// TIA Portal project "conveyor-push-sort" (V19)

(* hardware
DEVICE "S7-1200 station_1"  S7-1200 Station
   slot 0: "Rack_0"  S7-1200 Rack  Rack  V1.0
   slot 1: "PLC_1"  CPU 1214C AC/DC/Rly  6ES7 214-1BG40-0XB0  V4.2
   slot 3: "AQ 1x12BIT_1"  AQ1 signal board  6ES7 232-4HA30-0XB0  V1.0
*)

// ===== PLC "PLC_1"  CPU 1214C AC/DC/Rly =====

VAR_GLOBAL   // PLC tag table "Default tag table"
   "M_Start_LastState_Negative" AT %M11.1 : Bool;
   "M_Running" AT %M11.3 : Bool;
   "M_Push" AT %M11.4 : Bool;
   "M_Start_OneShot_Negative" AT %M11.2 : Bool;
   "M_MetalSensor_LastState_Positive" AT %M11.5 : Bool;
END_VAR

VAR_GLOBAL   // PLC tag table "ConveyorInput"
   "B1_FeederRetracted" AT %I0.2 : Bool;
   "B2_FeederExtended" AT %I0.3 : Bool;
   "B5_ColorSensor_IsWhite" AT %I0.6 : Bool;
   "B6_AtConveyorEnd" AT %I0.7 : Bool;
   "B4_MetalSensor" AT %I0.4 : Bool;
END_VAR

VAR_GLOBAL   // PLC tag table "ConveyorOutput"
   "Y1A_FeederExtend" AT %Q0.3 : Bool;
   "Y1B_FeederRetract" AT %Q0.2 : Bool;
   "B3_PusherRetracted" AT %I0.5 : Bool;
   "M1_ConveyorMove" AT %Q0.4 : Bool;
   "Y2_PusherExtend" AT %Q0.5 : Bool;
END_VAR

VAR_GLOBAL   // PLC tag table "ArmInput"
   "B8_ArmOverTruck" AT %I1.0 : Bool;
   "B7_ArmOverConveyor" AT %I1.1 : Bool;
   "B9_ArmIsDown" AT %I1.2 : Bool;
END_VAR

VAR_GLOBAL   // PLC tag table "OperatorPanel"
   "S1_Start" AT %I0.0 : Bool;   // NO
   "S2_Stop" AT %I0.1 : Bool;   // NO
   "P1_LightGreen" AT %Q0.0 : Bool;
   "P2_LightYellow" AT %Q0.1 : Bool;
END_VAR

VAR_GLOBAL   // PLC tag table "ArmOutput"
   "Y6_ArmFromTruckToConveyor" AT %Q0.6 : Bool;
   "Y4_LowerArm" AT %Q0.7 : Bool;
   "Y5_GripperPressureOn" AT %Q1.0 : Bool;
   "Y3_EnableBlackTruck" AT %Q1.1 : Bool;
   "B10_WhiteTruckActive" AT %I1.3 : Bool;
END_VAR

TYPE "ItemRecord"
   STRUCT
      AccumulatedTime : Time;
      Active : Bool;
   END_STRUCT;
END_TYPE

DATA_BLOCK "DB_Settings"   // DB2
{ S7_Optimized_Access := 'TRUE' }
VERSION : 0.1
   VAR
      FeederDelay : Time := T#100ms;
      ArmPickDelay : Time := T#120ms;
      ArmPlaceDelay : Time := T#200ms;
   END_VAR
BEGIN
END_DATA_BLOCK

DATA_BLOCK "DB_ArmSafeStopSteps"   // DB5
{ S7_Optimized_Access := 'TRUE' }
VERSION : 0.1
   VAR
      MovedOverConveyor : Bool;
      Lowered : Bool;
      Released : Bool;
      Lifted : Bool;
   END_VAR
BEGIN
END_DATA_BLOCK

DATA_BLOCK "DB_ItemTracking"   // DB6
{ S7_Optimized_Access := 'TRUE' }
VERSION : 0.1
   VAR
      ItemList : Array[0..5] of "ItemRecord";
      PrevScanTime : DTL;
      CurrentTime : DTL;
      DeltaTime : Time;
      UntrackedItems : UInt;
      ThresholdTime : Time := T#700ms;
   END_VAR
BEGIN
END_DATA_BLOCK

// folder: System blocks/Program resources

DATA_BLOCK "IEC_Timer_0_DB"   // DB1
{ S7_Optimized_Access := 'TRUE' }
AUTHOR : Simatic
FAMILY : IEC
NAME : IEC_TMR
VERSION : 1.0
// stored: InstanceOfName IEC_TIMER
"IEC_TIMER"
BEGIN
END_DATA_BLOCK

DATA_BLOCK "IEC_Timer_0_DB_1"   // DB3
{ S7_Optimized_Access := 'TRUE' }
AUTHOR : Simatic
FAMILY : IEC
NAME : IEC_TMR
VERSION : 1.0
// stored: InstanceOfName IEC_TIMER
"IEC_TIMER"
BEGIN
END_DATA_BLOCK

DATA_BLOCK "IEC_Timer_0_DB_3"   // DB4
{ S7_Optimized_Access := 'TRUE' }
AUTHOR : Simatic
FAMILY : IEC
NAME : IEC_TMR
VERSION : 1.0
// stored: InstanceOfName IEC_TIMER
"IEC_TIMER"
BEGIN
END_DATA_BLOCK

DATA_BLOCK "IEC_Timer_0_DB_2"   // DB7
{ S7_Optimized_Access := 'TRUE' }
AUTHOR : Simatic
FAMILY : IEC
NAME : IEC_TMR
VERSION : 1.0
// stored: InstanceOfName IEC_TIMER
"IEC_TIMER"
BEGIN
END_DATA_BLOCK

// folder: (top level)

FUNCTION "FC_Conveyor" : Void   // FC1, LAD
{ S7_Optimized_Access := 'TRUE' }
VERSION : 0.1
   VAR_TEMP
      i : Int;
      err : Int;
      CurrentTime : DTL;
   END_VAR
   VAR_TEMP   // added for the SCL form of the ladder/FBD networks
      _w1 : Bool;
   END_VAR
BEGIN

REGION Network 1 (SCL)
   // Track items
   IF "DB_ItemTracking".UntrackedItems > 0 THEN
       FOR #i := 0 TO 5 DO
           IF NOT "DB_ItemTracking".ItemList[#i].Active THEN
               "DB_ItemTracking".ItemList[#i].Active := TRUE;
               "DB_ItemTracking".UntrackedItems := "DB_ItemTracking".UntrackedItems - 1;
           END_IF;

           // If more items remain untracked, continue filling slots
           IF "DB_ItemTracking".UntrackedItems = 0 THEN
               EXIT;
           END_IF;
       END_FOR;
   END_IF;
END_REGION

REGION Network 2 (SCL)
   // Push items that approach pusher based on travel time
   #err := RD_SYS_T("DB_ItemTracking".CurrentTime);

   "DB_ItemTracking".DeltaTime := T_DIFF(IN1:="DB_ItemTracking".CurrentTime,IN2:="DB_ItemTracking".PrevScanTime);
   "DB_ItemTracking".PrevScanTime := "DB_ItemTracking".CurrentTime;

   IF "M1_ConveyorMove" THEN
       FOR #i := 0 TO 5 DO
           IF "DB_ItemTracking".ItemList[#i].Active THEN

               "DB_ItemTracking".ItemList[#i].AccumulatedTime :=
               "DB_ItemTracking".ItemList[#i].AccumulatedTime + "DB_ItemTracking".DeltaTime;

               IF "DB_ItemTracking".ItemList[#i].AccumulatedTime >= "DB_ItemTracking".ThresholdTime THEN
                   "M_Push" := TRUE;
                   "DB_ItemTracking".ItemList[#i].Active := FALSE;
                   "DB_ItemTracking".ItemList[#i].AccumulatedTime := T#0s;
               END_IF;
           END_IF;
       END_FOR;
   END_IF;
END_REGION

REGION Network 3
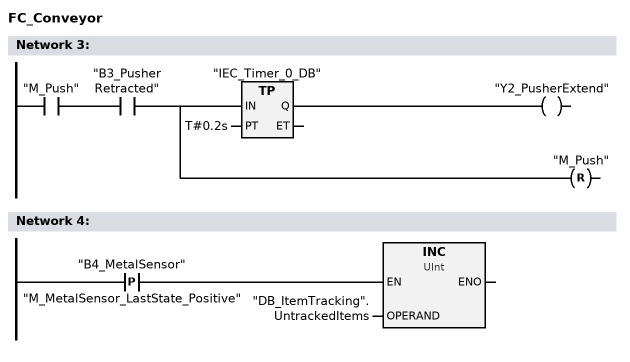
   #_w1 := "M_Push" AND "B3_PusherRetracted";
   "IEC_Timer_0_DB".TP(IN := #_w1, PT := T#0.2s);
   "Y2_PusherExtend" := "IEC_Timer_0_DB".Q;
   IF #_w1 THEN "M_Push" := FALSE; END_IF;
END_REGION

REGION Network 4
   RUNG wire#powerrail
      P_Contact(operand := "B4_MetalSensor", bit := "M_MetalSensor_LastState_Positive")
      { S7_Templates := "DestType := UInt" } Inc( "DB_ItemTracking".UntrackedItems )
   END_RUNG
   // the same network as SCL:
   #_w1 := "B4_MetalSensor" AND NOT "M_MetalSensor_LastState_Positive";   // rising edge of "B4_MetalSensor"
   "M_MetalSensor_LastState_Positive" := "B4_MetalSensor";
   IF #_w1 THEN "DB_ItemTracking".UntrackedItems := "DB_ItemTracking".UntrackedItems + 1; END_IF;
END_REGION
END_FUNCTION

FUNCTION "FC_Feeder" : Void   // FC2, LAD
{ S7_Optimized_Access := 'TRUE' }
VERSION : 0.1
BEGIN

REGION Network 1
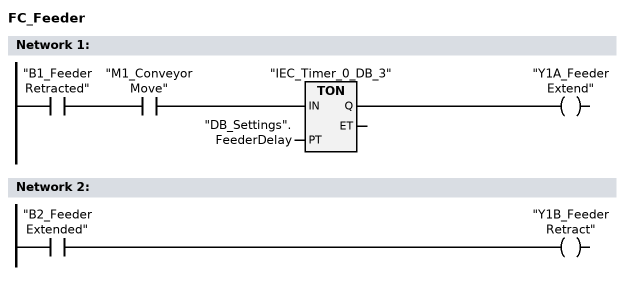
   "IEC_Timer_0_DB_3".TON(IN := "B1_FeederRetracted" AND "M1_ConveyorMove", PT := "DB_Settings".FeederDelay);
   "Y1A_FeederExtend" := "IEC_Timer_0_DB_3".Q;
END_REGION

REGION Network 2
   RUNG wire#powerrail
      Contact( "B2_FeederExtended" )
      Coil( "Y1B_FeederRetract" )
   END_RUNG
   // the same network as SCL:
   "Y1B_FeederRetract" := "B2_FeederExtended";
END_REGION
END_FUNCTION

FUNCTION "FC_PickAndPlace" : Void   // FC3, LAD
{ S7_Optimized_Access := 'TRUE' }
VERSION : 0.1
   VAR_TEMP   // added for the SCL form of the ladder/FBD networks
      _w1 : Bool;
      _w2 : Bool;
      _w3 : Bool;
   END_VAR
BEGIN

REGION Network 1
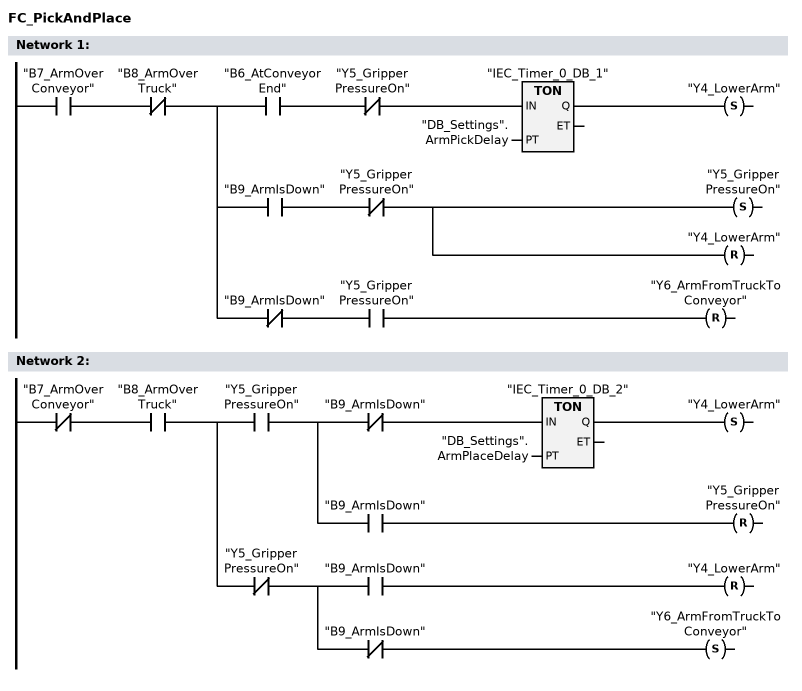
   #_w1 := "B7_ArmOverConveyor" AND NOT "B8_ArmOverTruck";
   "IEC_Timer_0_DB_1".TON(IN := #_w1 AND "B6_AtConveyorEnd" AND NOT "Y5_GripperPressureOn",
                          PT := "DB_Settings".ArmPickDelay);
   IF "IEC_Timer_0_DB_1".Q THEN "Y4_LowerArm" := TRUE; END_IF;
   #_w2 := #_w1 AND "B9_ArmIsDown" AND NOT "Y5_GripperPressureOn";
   IF #_w2 THEN
       "Y5_GripperPressureOn" := TRUE;
       "Y4_LowerArm" := FALSE;
   END_IF;
   IF #_w1 AND NOT "B9_ArmIsDown" AND "Y5_GripperPressureOn" THEN
       "Y6_ArmFromTruckToConveyor" := FALSE;
   END_IF;
END_REGION

REGION Network 2
   #_w1 := NOT "B7_ArmOverConveyor" AND "B8_ArmOverTruck";
   #_w2 := #_w1 AND "Y5_GripperPressureOn";
   "IEC_Timer_0_DB_2".TON(IN := #_w2 AND NOT "B9_ArmIsDown", PT := "DB_Settings".ArmPlaceDelay);
   IF "IEC_Timer_0_DB_2".Q THEN "Y4_LowerArm" := TRUE; END_IF;
   IF #_w2 AND "B9_ArmIsDown" THEN "Y5_GripperPressureOn" := FALSE; END_IF;
   #_w3 := #_w1 AND NOT "Y5_GripperPressureOn";
   IF #_w3 AND "B9_ArmIsDown" THEN "Y4_LowerArm" := FALSE; END_IF;
   IF #_w3 AND NOT "B9_ArmIsDown" THEN "Y6_ArmFromTruckToConveyor" := TRUE; END_IF;
END_REGION
END_FUNCTION

FUNCTION "FC_Truck" : Void   // FC4, LAD
{ S7_Optimized_Access := 'TRUE' }
VERSION : 0.1
   VAR_TEMP   // added for the SCL form of the ladder/FBD networks
      _w1 : Bool;
   END_VAR
BEGIN

REGION Network 1
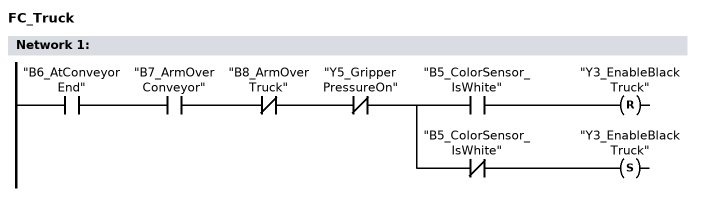
   RUNG wire#powerrail
      Contact( "B6_AtConveyorEnd" )
      Contact( "B7_ArmOverConveyor" )
      I_Contact( "B8_ArmOverTruck" )
      I_Contact( "Y5_GripperPressureOn" )
      wire#w1
      Contact( "B5_ColorSensor_IsWhite" )
      R_Coil( "Y3_EnableBlackTruck" )
   END_RUNG
   RUNG wire#w1
      I_Contact( "B5_ColorSensor_IsWhite" )
      S_Coil( "Y3_EnableBlackTruck" )
   END_RUNG
   // the same network as SCL:
   #_w1 := "B6_AtConveyorEnd" AND "B7_ArmOverConveyor" AND NOT "B8_ArmOverTruck" AND NOT "Y5_GripperPressureOn";
   IF #_w1 AND "B5_ColorSensor_IsWhite" THEN "Y3_EnableBlackTruck" := FALSE; END_IF;
   IF #_w1 AND NOT "B5_ColorSensor_IsWhite" THEN "Y3_EnableBlackTruck" := TRUE; END_IF;
END_REGION
END_FUNCTION

FUNCTION "FC_ArmSafeStop" : Void   // FC5, LAD
{ S7_Optimized_Access := 'TRUE' }
VERSION : 0.1
// One time executes actions required to set arm in a neutral position without the item over conveyor
   VAR_TEMP   // added for the SCL form of the ladder/FBD networks
      _w1 : Bool;
      _w2 : Bool;
   END_VAR
BEGIN

REGION Network 1
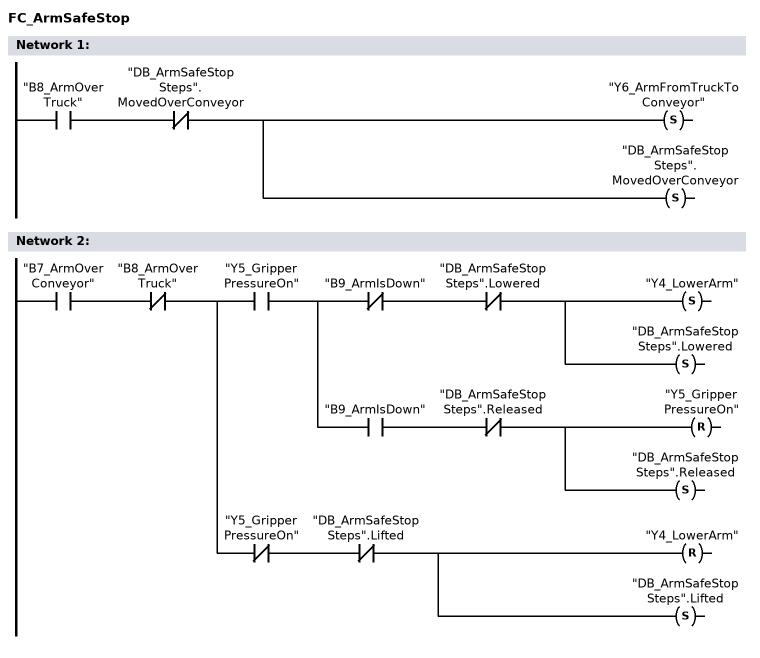
   RUNG wire#powerrail
      Contact( "B8_ArmOverTruck" )
      I_Contact( "DB_ArmSafeStopSteps".MovedOverConveyor )
      wire#w1
      S_Coil( "Y6_ArmFromTruckToConveyor" )
   END_RUNG
   RUNG wire#w1
      S_Coil( "DB_ArmSafeStopSteps".MovedOverConveyor )
   END_RUNG
   // the same network as SCL:
   IF "B8_ArmOverTruck" AND NOT "DB_ArmSafeStopSteps".MovedOverConveyor THEN
       "Y6_ArmFromTruckToConveyor" := TRUE;
       "DB_ArmSafeStopSteps".MovedOverConveyor := TRUE;
   END_IF;
END_REGION

REGION Network 2
   RUNG wire#powerrail
      Contact( "B7_ArmOverConveyor" )
      I_Contact( "B8_ArmOverTruck" )
      wire#w1
      Contact( "Y5_GripperPressureOn" )
      wire#w2
      I_Contact( "B9_ArmIsDown" )
      I_Contact( "DB_ArmSafeStopSteps".Lowered )
      wire#w3
      S_Coil( "Y4_LowerArm" )
   END_RUNG
   RUNG wire#w3
      S_Coil( "DB_ArmSafeStopSteps".Lowered )
   END_RUNG
   RUNG wire#w2
      Contact( "B9_ArmIsDown" )
      I_Contact( "DB_ArmSafeStopSteps".Released )
      wire#w4
      R_Coil( "Y5_GripperPressureOn" )
   END_RUNG
   RUNG wire#w4
      S_Coil( "DB_ArmSafeStopSteps".Released )
   END_RUNG
   RUNG wire#w1
      I_Contact( "Y5_GripperPressureOn" )
      I_Contact( "DB_ArmSafeStopSteps".Lifted )
      wire#w5
      R_Coil( "Y4_LowerArm" )
   END_RUNG
   RUNG wire#w5
      S_Coil( "DB_ArmSafeStopSteps".Lifted )
   END_RUNG
   // the same network as SCL:
   #_w1 := "B7_ArmOverConveyor" AND NOT "B8_ArmOverTruck";
   #_w2 := #_w1 AND "Y5_GripperPressureOn";
   IF #_w2 AND NOT "B9_ArmIsDown" AND NOT "DB_ArmSafeStopSteps".Lowered THEN
       "Y4_LowerArm" := TRUE;
       "DB_ArmSafeStopSteps".Lowered := TRUE;
   END_IF;
   IF #_w2 AND "B9_ArmIsDown" AND NOT "DB_ArmSafeStopSteps".Released THEN
       "Y5_GripperPressureOn" := FALSE;
       "DB_ArmSafeStopSteps".Released := TRUE;
   END_IF;
   IF #_w1 AND NOT "Y5_GripperPressureOn" AND NOT "DB_ArmSafeStopSteps".Lifted THEN
       "Y4_LowerArm" := FALSE;
       "DB_ArmSafeStopSteps".Lifted := TRUE;
   END_IF;
END_REGION
END_FUNCTION

ORGANIZATION_BLOCK "Main"   // OB1, LAD, ProgramCycle
TITLE = "Main Program Sweep (Cycle)"
{ S7_Optimized_Access := 'TRUE' }
VERSION : 0.1
   VAR_INPUT
      Initial_Call : Bool;   // Initial call of this OB
      Remanence : Bool;   // =True, if remanent data are available
   END_VAR
   VAR_TEMP   // added for the SCL form of the ladder/FBD networks
      _w1 : Bool;
   END_VAR
BEGIN

REGION Network 1
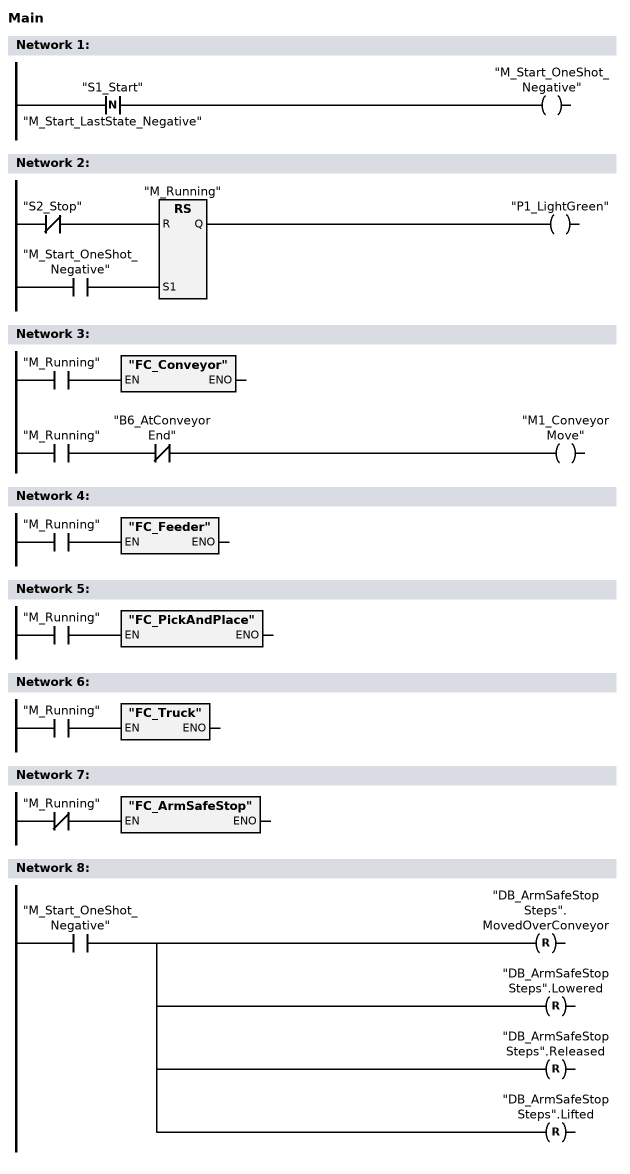
   RUNG wire#powerrail
      N_Contact(operand := "S1_Start", bit := "M_Start_LastState_Negative")
      Coil( "M_Start_OneShot_Negative" )
   END_RUNG
   // the same network as SCL:
   #_w1 := NOT "S1_Start" AND "M_Start_LastState_Negative";   // falling edge of "S1_Start"
   "M_Start_LastState_Negative" := "S1_Start";
   "M_Start_OneShot_Negative" := #_w1;
END_REGION

REGION Network 2
   RUNG wire#powerrail
      I_Contact( "S2_Stop" )
      S_RS(operand := "M_Running", s1 := wire#w1)
      Coil( "P1_LightGreen" )
   END_RUNG
   RUNG wire#powerrail
      Contact( "M_Start_OneShot_Negative" )
   END_RUNG wire#w1
   // the same network as SCL:
   IF NOT "S2_Stop" THEN
       "M_Running" := FALSE;   // RS flip-flop
   END_IF;
   IF "M_Start_OneShot_Negative" THEN "M_Running" := TRUE; END_IF;
   "P1_LightGreen" := "M_Running";
END_REGION

REGION Network 3
   RUNG wire#powerrail
      Contact( "M_Running" )
      "FC_Conveyor"()
   END_RUNG
   RUNG wire#powerrail
      Contact( "M_Running" )
      I_Contact( "B6_AtConveyorEnd" )
      Coil( "M1_ConveyorMove" )
   END_RUNG
   // the same network as SCL:
   IF "M_Running" THEN "FC_Conveyor"(); END_IF;
   "M1_ConveyorMove" := "M_Running" AND NOT "B6_AtConveyorEnd";
END_REGION

REGION Network 4
   RUNG wire#powerrail
      Contact( "M_Running" )
      "FC_Feeder"()
   END_RUNG
   // the same network as SCL:
   IF "M_Running" THEN "FC_Feeder"(); END_IF;
END_REGION

REGION Network 5
   RUNG wire#powerrail
      Contact( "M_Running" )
      "FC_PickAndPlace"()
   END_RUNG
   // the same network as SCL:
   IF "M_Running" THEN "FC_PickAndPlace"(); END_IF;
END_REGION

REGION Network 6
   RUNG wire#powerrail
      Contact( "M_Running" )
      "FC_Truck"()
   END_RUNG
   // the same network as SCL:
   IF "M_Running" THEN "FC_Truck"(); END_IF;
END_REGION

REGION Network 7
   RUNG wire#powerrail
      I_Contact( "M_Running" )
      "FC_ArmSafeStop"()
   END_RUNG
   // the same network as SCL:
   IF NOT "M_Running" THEN "FC_ArmSafeStop"(); END_IF;
END_REGION

REGION Network 8
   RUNG wire#powerrail
      Contact( "M_Start_OneShot_Negative" )
      wire#w1
      R_Coil( "DB_ArmSafeStopSteps".MovedOverConveyor )
   END_RUNG
   RUNG wire#w1
      R_Coil( "DB_ArmSafeStopSteps".Lowered )
   END_RUNG
   RUNG wire#w1
      R_Coil( "DB_ArmSafeStopSteps".Released )
   END_RUNG
   RUNG wire#w1
      R_Coil( "DB_ArmSafeStopSteps".Lifted )
   END_RUNG
   // the same network as SCL:
   IF "M_Start_OneShot_Negative" THEN
       "DB_ArmSafeStopSteps".MovedOverConveyor := FALSE;
       "DB_ArmSafeStopSteps".Lowered := FALSE;
       "DB_ArmSafeStopSteps".Released := FALSE;
       "DB_ArmSafeStopSteps".Lifted := FALSE;
   END_IF;
END_REGION
END_ORGANIZATION_BLOCK